FUNCTION_BLOCK CamTable IMPLEMENTS itfCamTable
VAR_INPUT
END_VAR
VAR_OUTPUT
END_VAR
VAR
END_VAR

{warning 'Add method implementation '}
METHOD Select		: itfCommand
VAR_INPUT
	Periodic		: BOOL;
	MasterAbsolute	: BOOL;
	SlaveAbsolute	: BOOL;
	CamTable		: MC_CAM_REF;
END_VAR
END_METHOD

END_FUNCTION_BLOCK

(* stored: Version 1.1.0.1, ProductVersion 3.1.4024.12
   POU CamTable: Id {4dbc9424-92e7-42bb-89db-96e536f03565}, SpecialFunc None
   Method Select: Id {f267f0fd-b892-4adb-818b-5335e87f5f6e} *)
